INTERFACE Motor

METHOD AanUit
VAR_INPUT
END_VAR
END_METHOD

END_INTERFACE

(* stored: Version 1.1.0.1
   Itf Motor: Id {d3f47777-bd5b-48b1-bdcb-ea49bd88495e}
   Method AanUit: Id {060d63f9-787c-496d-9022-28764b8b1e72} *)
